// TIA Portal V20 export
DATA_BLOCK "Receive_FData_DB"   // DB4
// stored: InstanceOfName Receive_FData, InstanceOfType FB
"Receive_FData"
   // VAR
   //    TRCV_Instance { S7_SetPoint := 'True'} : TRCV;
   // END_VAR
BEGIN
END_DATA_BLOCK
